// TwinCAT 3 PLC project PLC_ImageStatistics
// ProgramVersion: 3.1.4024.12
// libraries:
//   Tc2_Standard, * (Beckhoff Automation GmbH)
//   Tc2_System, * (Beckhoff Automation GmbH)
//   Tc2_Utilities, * (Beckhoff Automation GmbH)
//   Tc3_Module, * (Beckhoff Automation GmbH)
//   Tc3_Vision, * (Beckhoff Automation GmbH)
// project tree:
//   / PlcTask.TcTTO
//   POUs/ MAIN.TcPOU
// real-time tasks:
//   TASK PlcTask: cycle T#10ms, priority 20, ADS port 350
//   TASK VnTask ImgAcq (FileSource1): cycle T#10ms, priority 5, ADS port 351

CONFIGURATION PLC_ImageStatistics
    RESOURCE PLC ON TwinCAT3
        TASK PlcTask(INTERVAL := T#10ms, PRIORITY := 20);
        PROGRAM MAIN WITH PlcTask : MAIN;
    END_RESOURCE
END_CONFIGURATION

// ---- POUs/MAIN.TcPOU
PROGRAM MAIN
VAR
	hr				:	HRESULT;
	ipImageIn		:	ITcVnImage;
	ipImageInDisp	:	ITcVnDisplayableImage;
	ipImageRes		:	ITcVnImage;
	ipImageResDisp	:	ITcVnDisplayableImage;
	fbCameraControl	:	FB_VN_SimpleCameraControl;
	eCameraState	:	ETcVnCameraState;
	stImageInfo		:	TcVnImageInfo;
	
	aMin			:	TcVnVector4_LREAL;
	aMax			:	TcVnVector4_LREAL;
	aMedian			:	TcVnVector4_LREAL;
	aAverage		:	TcVnVector4_LREAL;
	aStdDev			:	TcVnVector4_LREAL;
	
	aPos			:	TcVnPoint2_DINT;
	sText			:	STRING;
	
	nTextX			:	UDINT	:=	10;
	nTextYBase		:	UDINT	:=	50;
	nTextYIncrement	:	UDINT	:=	50;
	fFontScale		:	LREAL	:=	2;
END_VAR

//	Disclaimer
  	
//	THIS publication contains statements about the suitability OF our products FOR certain 
//	areas OF application. These statements are based on typical features OF our products. 
//	The examples shown in THIS publication are FOR demonstration purposes only. The 
//	information provided herein should NOT be regarded as specific operation characteristics. 
//	It is incumbent on the customer TO check AND decide whether a product is suitable FOR use 
//	in a particular application. We DO NOT give ANY warranty that the source code which is 
//	made available with this publication is complete or accurate. 
  	
//	THE SAMPLE CODE CONTAINED IN THIS PUBLICATION IS PROVIDED “AS IS” WITHOUT WARRANTY OF ANY 
//	KIND, EITHER EXPRESSED, IMPLIED OR STATUTORY, INCLUDING WITHOUT LIMITATION, ANY WARRANTY 
//	WITH RESPECT TO NON-INFRINGEMENT, FREEDOM FROM PROPRIETARY RIGHTS OF THIRD PARTIES OR 
//	FITNESS FOR ANY PARTICULAR PURPOSE. 
  	
//	THIS publication may be changed FROM TIME TO TIME without prior notice. No liability 
//	is assumed FOR errors AND/OR omissions. Our products are described in detail in our 
//	data sheets AND documentations. Product-specific warnings AND cautions must be observed. 
//	FOR the latest version OF our data sheets AND documentations visit our website 
//	(www.beckhoff.de). 
  	
//	© Beckhoff Automation GmbH & Co. KG, March 2020
  	
//	The reproduction, distribution AND utilization OF THIS document as well as the 
//	communication OF its contents TO others without express authorization is prohibited. 
//	Offenders will be held liable FOR the payment OF damages. All rights reserved in the 
//	event of the grant of a patent, utility model or design.

//	==========================================================================================

//	Sample: Image Statistics
//	----------------------------------------

//	Steps to do:
//	 1. Add images to the FileSource1

eCameraState := fbCameraControl.GetState();

// CameraControl is in error state, so try to reset the camera connection
IF eCameraState = TCVN_CS_ERROR THEN
	hr := fbCameraControl.Reset();

// Camera not yet streaming
ELSIF eCameraState < TCVN_CS_ACQUIRING THEN
	hr := fbCameraControl.StartAcquisition();

// Camera streaming
ELSIF eCameraState = TCVN_CS_ACQUIRING THEN
	hr := fbCameraControl.GetCurrentImage(ipImageIn);
	
	IF SUCCEEDED(hr) AND ipImageIn <> 0 THEN
		
		// Input validation and prepare images
		hr := F_VN_GetImageInfo(ipImageIn, stImageInfo, hr);
		IF stImageInfo.stPixelFormat.nChannels = 1 THEN
			; // right type, no conversion needed 
		ELSIF stImageInfo.stPixelFormat.nChannels = 3 THEN
			hr := F_VN_ConvertColorSpace(ipImageIn, ipImageIn, TCVN_CST_RGB_TO_GRAY, hr);
		ELSIF stImageInfo.stPixelFormat.nChannels = 4 THEN
			hr := F_VN_ConvertColorSpace(ipImageIn, ipImageIn, TCVN_CST_RGBA_TO_GRAY, hr);
		ELSE
			hr := Tc2_System.E_HRESULTAdsErr.INCOMPATIBLE;
		END_IF
		
		hr := F_VN_CopyImage(ipImageIn, ipImageRes, hr);
		
		// Calculate image statistics
		hr := F_VN_MinPixelValue(
			ipImage		:=	ipImageIn,
			aMinValue	:=	aMin,
			aPosition	:=	aPos,
			hrPrev		:=	hr);
			
		hr := F_VN_MaxPixelValue(
			ipImage		:=	ipImageIn,
			aMaxValue	:=	aMax,
			aPosition	:=	aPos,
			hrPrev		:=	hr);
			
		hr := F_VN_ImageMedian(
			ipSrcImage	:=	ipImageIn,
			aMedian		:=	aMedian,
			hrPrev		:=	hr);
			
		hr := F_VN_ImageAverageStdDev(
			ipSrcImage	:=	ipImageIn,
			aAverage	:=	aAverage,
			aStdDev		:=	aStdDev,
			hrPrev		:=	hr);
		
		// Adjust font scale depending on image width
		IF stImageInfo.nWidth <= 500 THEN
			fFontScale := 1;
			nTextYIncrement := 25;
		ELSIF stImageInfo.nWidth <= 800 THEN
			fFontScale := 2;
			nTextYIncrement := 50;
		ELSE
			fFontScale := 3;
			nTextYIncrement := 75;
		END_IF
		
		// Draw results
		sText := CONCAT('Min: ', LREAL_TO_FMTSTR(aMin[0], 2, TRUE ));
		hr := F_VN_PutLabel(sText, ipImageRes, nTextX, (nTextYBase + (1 * nTextYIncrement)), fFontScale, hr);
		sText := CONCAT('Max: ', LREAL_TO_FMTSTR(aMax[0], 2, TRUE ));
		hr := F_VN_PutLabel(sText, ipImageRes, nTextX, (nTextYBase + (2 * nTextYIncrement)), fFontScale, hr);
		sText := CONCAT('Median: ', LREAL_TO_FMTSTR(aMedian[0], 2, TRUE ));
		hr := F_VN_PutLabel(sText, ipImageRes, nTextX, (nTextYBase + (3 * nTextYIncrement)), fFontScale, hr);
		sText := CONCAT('Average: ', LREAL_TO_FMTSTR(aAverage[0], 2, TRUE ));
		hr := F_VN_PutLabel(sText, ipImageRes, nTextX, (nTextYBase + (4 * nTextYIncrement)), fFontScale, hr);
		sText := CONCAT('StdDev: ', LREAL_TO_FMTSTR(aStdDev[0], 2, TRUE ));
		hr := F_VN_PutLabel(sText, ipImageRes, nTextX, (nTextYBase + (5 * nTextYIncrement)), fFontScale, hr);
		
		hr := F_VN_TransformIntoDisplayableImage(ipImageIn, ipImageInDisp, hr);
		hr := F_VN_TransformIntoDisplayableImage(ipImageRes, ipImageResDisp, hr);
	END_IF
END_IF

END_PROGRAM
